ABB RAPID module: Product1Mod.modx

MODULE Product1Mod



    PROC SeqProduct1()
        ProductPick;
        ProductProcess;
        ProductPlace;
    ENDPROC



    LOCAL PROC ProductPick()
        GripClose;
    ENDPROC



    LOCAL PROC ProductProcess()
        !
    ENDPROC



    LOCAL PROC ProductPlace()
        GripOpen;
    ENDPROC



    PROC ForgottenTestProc()
        !
    ENDPROC



ENDMODULE
